{attribute 'qualified_only'}
//{attribute 'strict'}
{attribute 'to_string'}
TYPE E_LogicIfCondition :
(
	PASS := 0,
	INPUT := 1,
	REGISTER := 2,
	COUNTER := 3
);
END_TYPE

(* stored: Version 1.1.0.1
   EnumerationTextList E_LogicIfCondition: Id {01764ae0-ed07-413e-b434-fbf743be9a29} *)
